FUNCTION_BLOCK FB_AlarmCalculator
VAR CONSTANT
	NUM_OF_SEVERITIES: INT  := 5;
	COMMAND_QUEUE_BUFFER_SIZE :INT := 20;
	NUM_OF_LISTENER: INT := 10;
END_VAR
VAR_INPUT
	bRefresh	: BOOL;			// make true at momentally (1 cycle) when 
END_VAR
VAR_OUTPUT
END_VAR
VAR
	al_index	: UINT := 0;
	p_alarms	: ARRAY [0..AlarmEventParam.ALARM_MAX_COUNT - 1] OF POINTER TO FB_Alarm;
	_listeners	: ARRAY [1..NUM_OF_LISTENER] OF I_Observer;
	//_p_exporter	: POINTER TO FB_AlarmDBExporter;
	state_counter	: ARRAY [0..NUM_OF_SEVERITIES - 1] OF EventSeverityStatusMember := [
		(severity := TcEventSeverity.Verbose),(severity := TcEventSeverity.Info),(severity := TcEventSeverity.Warning),
		(severity := TcEventSeverity.Error),(severity := TcEventSeverity.Critical)
	];
	_counter 	:UINT;
	i			: INT;
	j			: INT;
	
	
	// queue controll
	
	_queue_usage:	UDINT;
	_queue_size:	UDINT := COMMAND_QUEUE_BUFFER_SIZE;
	nWriteIndex: 	UDINT;
	nReadIndex: 	UDINT;
	queue_buffer:	ARRAY [0..COMMAND_QUEUE_BUFFER_SIZE - 1] OF PVOID;
	event_text:		STRING;
	pAlarm:			POINTER TO FB_Alarm;
	_lang_code:		DINT := 1031; 
	_step: UINT;
END_VAR

FOR j := 0 TO NUM_OF_SEVERITIES - 1 DO
	state_counter[j].active_counter := 0;
	state_counter[j].raised_counter := 0;
	state_counter[j].confirmed_counter := 0;		
END_FOR
FOR i := 0 TO al_index - 1 DO
	j := p_alarms[i]^.eSeverity;
	IF p_alarms[i]^.bEvt THEN
		state_counter[j].active_counter := state_counter[j].active_counter + 1;
	END_IF
	IF p_alarms[i]^.bActive THEN
		state_counter[j].raised_counter := state_counter[j].raised_counter + 1;
	END_IF
	IF p_alarms[i]^.bActive AND p_alarms[i]^.eConfirmationState <> TcEventConfirmationState.WaitForConfirmation THEN
		state_counter[j].confirmed_counter := state_counter[j].confirmed_counter + 1;
	END_IF
	IF p_alarms[i]^.event_raised OR p_alarms[i]^.event_cleared THEN
		put(p_alarms[i]);
	END_IF
END_FOR

CASE _step OF
	0 :
		IF _queue_usage > 0 THEN
			pAlarm := get();
			_step := 10;
		END_IF
	10:
		FOR i := 1 TO NUM_OF_LISTENER DO
			IF _listeners[i] <> 0 AND pAlarm <> 0 THEN
				IF pAlarm^.get_alarm_text(_lang_code) THEN
					_listeners[i].send_signal(pAlarm);
					_step := 0;
				END_IF
			END_IF			
		END_FOR
END_CASE

METHOD add_listener : INT
VAR_INPUT
	listener: I_Observer;
END_VAR
VAR
	i :INT;
END_VAR
add_listener := 0;
IF listener = 0 THEN
	RETURN;
END_IF

FOR i := 1 TO NUM_OF_LISTENER DO
	IF _listeners[i] = 0 THEN
		_listeners[i] := listener;
		add_listener := i;
		RETURN;
	END_IF
END_FOR
END_METHOD

METHOD clear_listners : BOOL
VAR_INPUT
END_VAR
VAR
	i : INT;
END_VAR
clear_listners := FALSE;
FOR i := 1 TO NUM_OF_LISTENER DO
	_listeners[i] := 0;
END_FOR
clear_listners := TRUE;
END_METHOD

PROPERTY full : BOOL
GET
full :=  _queue_usage >= COMMAND_QUEUE_BUFFER_SIZE - 1;
END_GET
END_PROPERTY

METHOD get : PVOID
VAR_INPUT
END_VAR
//Set buffer index

IF _queue_usage > 0 THEN
	get := queue_buffer[nReadIndex];
	_queue_usage := _queue_usage - 1;
	nReadIndex := nReadIndex + 1;
	IF nReadIndex > COMMAND_QUEUE_BUFFER_SIZE - 1 THEN
		nReadIndex := 0;
	END_IF
END_IF

RETURN;
END_METHOD

METHOD is_active : BOOL
VAR_INPUT
	severity : TcEventSeverity := TcEventSeverity.Error; // Filterd minimum serverity level
END_VAR
VAR
	i:	UINT;
END_VAR
is_active := FALSE;
FOR i := severity TO NUM_OF_SEVERITIES - 1 DO
	IF state_counter[i].active_counter > 0 THEN
		is_active := TRUE;
		RETURN;
	END_IF
END_FOR
END_METHOD

// TRUE if the registered events filtered by specified severity level is in Raised state.
METHOD PUBLIC is_raised : BOOL
VAR_INPUT
	severity : TcEventSeverity := TcEventSeverity.Error; // Filterd minimum serverity level
END_VAR
VAR
	i:	UINT;
END_VAR
is_raised := FALSE;
FOR i := severity TO NUM_OF_SEVERITIES - 1 DO
	IF state_counter[i].raised_counter > 0  THEN
		is_raised := TRUE;
		RETURN;
	END_IF
END_FOR
END_METHOD

// TRUE if the registered events filtered by specified severity level is in WaitForConfirmation state.
METHOD PUBLIC is_unconfirmed : BOOL
VAR_INPUT
	severity : TcEventSeverity := TcEventSeverity.Error; // Filterd minimum serverity level
END_VAR
VAR
	i:	UINT;
END_VAR
is_unconfirmed := FALSE;
FOR i := severity TO NUM_OF_SEVERITIES - 1 DO
	IF state_counter[i].raised_counter > state_counter[i].confirmed_counter THEN
		is_unconfirmed := TRUE;
		RETURN;
	END_IF
END_FOR
END_METHOD

{warning 'add property implementation'}
PROPERTY lang_code : DINT
GET
lang_code := _lang_code;
END_GET
SET
_lang_code := lang_code;
END_SET
END_PROPERTY

PROPERTY p_alarm_list : PVOID
GET
p_alarm_list := ADR(p_alarms);
END_GET
END_PROPERTY

METHOD put : BOOL
VAR_INPUT
	lData:	PVOID;
END_VAR
//Set buffer index

IF _queue_usage >= COMMAND_QUEUE_BUFFER_SIZE - 1 THEN
	put := 0;
ELSE
	queue_buffer[nWriteIndex] := lData;
	_queue_usage := _queue_usage + 1;
	nWriteIndex := nWriteIndex + 1;
	IF nWriteIndex > COMMAND_QUEUE_BUFFER_SIZE - 1 THEN
		nWriteIndex := 0;
	END_IF
	put := 1;
END_IF

RETURN;
END_METHOD

METHOD INTERNAL reg_alarm : BOOL
VAR_INPUT
	p_alarm	:POINTER TO FB_Alarm;
END_VAR
IF AlarmEventParam.ALARM_MAX_COUNT <= al_index THEN
	reg_alarm := FALSE;
	RETURN;
END_IF

p_alarms[al_index] := p_alarm;
al_index := al_index + 1;
reg_alarm := TRUE;
END_METHOD

METHOD rm_listener : INT
VAR_INPUT
	listener : I_Observer;
END_VAR
VAR
	i : INT;
END_VAR
rm_listener := 0;
IF listener = 0 THEN
	RETURN;
END_IF

FOR i := 1 TO NUM_OF_LISTENER DO
	IF _listeners[i] = listener THEN
		_listeners[i] := 0;
		rm_listener := i;
		RETURN;
	END_IF
END_FOR
END_METHOD

END_FUNCTION_BLOCK

(* stored: Version 1.1.0.1, ProductVersion 3.1.4024.12
   POU FB_AlarmCalculator: Id {f9fb4732-2a58-4724-8e9e-37487e3bcd05}, SpecialFunc None
   Method add_listener: Id {8921ab30-f5c2-4c4b-994e-23daf3905bf7}
   Method clear_listners: Id {ef54ad0c-c9b9-4e2f-92f1-349b1e4d19d3}
   Property full: Id {e3de9c67-ef8c-4885-b0d0-c9c6d8211ff9}
   Get Get: Id {f87d1f5c-efdd-40b1-a1b7-dd2f20e9ba27}
   Method get: Id {7d30b5e5-3cde-4ac8-bc75-313862a9fcfc}
   Method is_active: Id {07aa9bb9-d63a-4e70-ac95-7d6d764146f1}
   Method is_raised: Id {de96aac9-c9b2-4695-bd6f-841b669f2da8}
   Method is_unconfirmed: Id {154448da-2a54-4ab5-b3d4-96a70c7c1c3e}
   Property lang_code: Id {d16b24d8-fc6b-4de5-9635-69e1c70a5846}
   Get Get: Id {b97d26d3-ff91-4b2a-9bf0-bbb8f21df6ee}
   Set Set: Id {722ab80b-bb02-4b63-ae92-426a8a494104}
   Property p_alarm_list: Id {90b2eb37-4f2f-48cd-82d9-aa401f30f999}
   Get Get: Id {8820ab56-5de6-4761-96ff-2c635d634b8c}
   Method put: Id {93203208-f677-42c4-9276-d0f7d8d17596}
   Method reg_alarm: Id {9282b111-287e-4a69-a8d7-7357a254d643}
   Method rm_listener: Id {6dd38a8c-f36d-42a8-ae40-3779706ac0f0} *)
